(* PLC project Thermal Control, Unknown Unnamed 1 *)
(* stored: creationDateTime 2025-10-18T00:08:59, modificationDateTime 2025-10-18T00:19:27 *)

PROGRAM thermal_control_ST
  VAR
    Temperature AT %IW100 : INT;  (* Temperature input from Modbus (K × 100) *)
  END_VAR
  VAR
    HeaterFeedback AT %IW101 : INT;  (* Heater state feedback: 0=OFF, 100=ON *)
  END_VAR
  VAR
    HeaterCommand AT %QX0.0 : BOOL;  (* Output to control heater coil *)
  END_VAR
  VAR
    TempLow : INT;  (* Low threshold: 291.15 K (18°C) *)
    TempHigh : INT;  (* High threshold: 295.15 K (22°C) *)
  END_VAR

            TempLow := 29115;
TempHigh := 29515;

IF Temperature < TempLow THEN
    HeaterCommand := TRUE;
ELSIF Temperature > TempHigh THEN
    HeaterCommand := FALSE;
END_IF;
          
END_PROGRAM

PROGRAM heater_on_ST
  VAR
    HeaterCommand AT %QX0.0 : BOOL;  (* Output to control heater *)
  END_VAR

            HeaterCommand := TRUE;
          
END_PROGRAM

PROGRAM read_temp_ST
  VAR
    Temperature AT %IW100 : INT;  (* Temperature input from Modbus *)
  END_VAR
  VAR
    TempDisplayed : INT;  (* Copy for monitoring *)
  END_VAR

            TempDisplayed := Temperature;
          
END_PROGRAM

CONFIGURATION Config0
  RESOURCE Res0 ON PLC
    TASK task0(INTERVAL := T#20ms, PRIORITY := 0);
    PROGRAM instance0 WITH task0 : thermal_control_ST;
  END_RESOURCE
END_CONFIGURATION
